// SIMATIC STEP 7 (V5.x) project KURS_PLC
// CPU: CPU 319-3 PN/DP
// station: Hardware
// station: SIMATIC 300(1)
// station: P_ADR_BUS
// program: S7 Program(2)

SYMBOL_TABLE
"SIM_M1"	DB 1	FB 1	// simulation: motor 1
"SIM_CONSTANS"	DB 2	DB 2	// simulation constants
"SIM_M"	FB 1	FB 1	// simulation: electric motor
"SIM_TANK"	FB 20	FB 20	// simulation: tank
"SIM"	FC 1	FC 1	// simulation environment
"U_TANK"	FC 20	FC 20
"h_level"	FC 21	FC 21
"U_HEAT"	FC 22	FC 22
"U_COOL"	FC 23	FC 23
"Ca"	FC 24	FC 24
"TANK"	FC 25	FC 25
"CTRL_MOTOR_SIMPLE"	FC 101	FC 101	// electric motor control
"TEST_MOTOR"	FC 1001	FC 1001	// test: CTRL_MOTOR_SIMPLE
"M1.ON"	M 1.0	BOOL
"M1.RUN"	M 1.1	BOOL
"M1.ALARM"	M 1.2	BOOL
"M1.ALARMM"	M 1.3	BOOL
"M1.RESET"	M 1.4	BOOL
"M1.CTRL"	M 1.5	BOOL
"VIN1.OPEN"	M 2.0	BOOL
"VIN1.CLOSED"	M 2.1	BOOL
"VIN2.OPEN"	M 2.2	BOOL
"VIN2.CLOSED"	M 2.3	BOOL
"k_IN1"	M 2.4	BOOL
"k_IN2"	M 2.5	BOOL
"SIM_START"	M 3.0	BOOL
"SIM_RESET"	M 3.1	BOOL
"k_HEAT"	MD 4	REAL
"k_COOL"	MD 8	REAL
"k_OUT"	MD 12	REAL
"U_COOLIN"	MD 16	REAL
"U_HEATIN"	MD 20	REAL
"U_IN2"	MD 24	REAL
"Ca_IN2"	MD 28	REAL
"U_IN1"	MD 32	REAL
"Ca_IN1"	MD 36	REAL
"Q_IN1"	MD 40	REAL
"Q_IN2"	MD 44	REAL
"SIMULATION"	OB 35	OB 35
"SRT_DINT"	SFC 32	SFC 32	// Start Time-Delay Interrupt
"QRY_DINT"	SFC 34	SFC 34	// Query Time-Delay Interrupt
"SIM_TEST"	VAT 1		// simulation test
END_SYMBOL_TABLE

FUNCTION_BLOCK "SIM_M"	// FB 1
TITLE = simulation: electric motor
//Uproszczony model silnika elektrycznego
//stany:
//STOP (0) - silnik wyłączony
//STARTING (1) - rozruch silnika
//RUN (2) - praca silnika
//STOPPING (3) - zatrzymanie silnika
VERSION : 0.1
VAR_INPUT
  On : BOOL ;	//zalaczenie silnika
  StartTime : INT ;	//czas rozruchu
  StopTime : INT ;	//czas zatrzymania
END_VAR
VAR_OUTPUT
  Run : BOOL ;
END_VAR
VAR
  State : INT ;	//numer stanu silnika
  Cnt : INT ;	//licznik czasu rozruchu/zatrzymania silnika
END_VAR
VAR_TEMP
  TempBool : BOOL ;
END_VAR
BEGIN
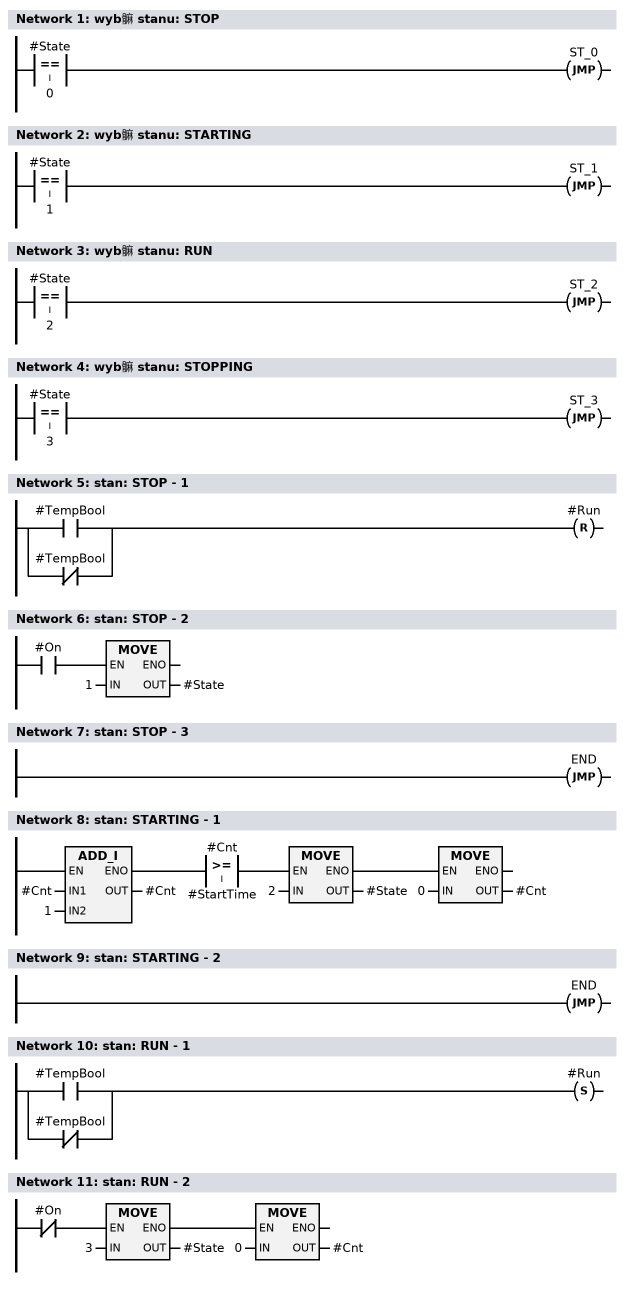
NETWORK
TITLE = wybór stanu: STOP
      L     #State;
      L     0;
      ==I;
      JC    ST_0;
NETWORK
TITLE = wybór stanu: STARTING
      L     #State;
      L     1;
      ==I;
      JC    ST_1;
NETWORK
TITLE = wybór stanu: RUN
      L     #State;
      L     2;
      ==I;
      JC    ST_2;
NETWORK
TITLE = wybór stanu: STOPPING
      L     #State;
      L     3;
      ==I;
      JC    ST_3;
NETWORK
TITLE = stan: STOP - 1
ST_0: O     #TempBool;
      ON    #TempBool;
      R     #Run;
NETWORK
TITLE = stan: STOP - 2
      A     #On;
      JNB   _001;
      L     1;
      T     #State;
_001: NOP   0;
NETWORK
TITLE = stan: STOP - 3
      JU    END;
NETWORK
TITLE = stan: STARTING - 1
ST_1: A(;
      A(;
      L     #Cnt;
      L     1;
      +I;
      T     #Cnt;
      AN    OV;
      SAVE;
      CLR;
      A     BR;
      );
      A(;
      L     #Cnt;
      L     #StartTime;
      >=I;
      );
      JNB   _002;
      L     2;
      T     #State;
      SET;
      SAVE;
      CLR;
_002: A     BR;
      );
      JNB   _003;
      L     0;
      T     #Cnt;
_003: NOP   0;
NETWORK
TITLE = stan: STARTING - 2
      JU    END;
NETWORK
TITLE = stan: RUN - 1
ST_2: O     #TempBool;
      ON    #TempBool;
      S     #Run;
NETWORK
TITLE = stan: RUN - 2
      A(;
      AN    #On;
      JNB   _004;
      L     3;
      T     #State;
      SET;
      SAVE;
      CLR;
_004: A     BR;
      );
      JNB   _005;
      L     0;
      T     #Cnt;
_005: NOP   0;
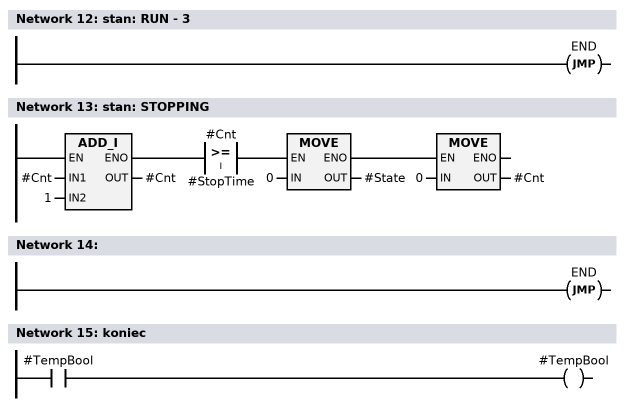
NETWORK
TITLE = stan: RUN - 3
      JU    END;
NETWORK
TITLE = stan: STOPPING
ST_3: A(;
      A(;
      L     #Cnt;
      L     1;
      +I;
      T     #Cnt;
      AN    OV;
      SAVE;
      CLR;
      A     BR;
      );
      A(;
      L     #Cnt;
      L     #StopTime;
      >=I;
      );
      JNB   _006;
      L     0;
      T     #State;
      SET;
      SAVE;
      CLR;
_006: A     BR;
      );
      JNB   _007;
      L     0;
      T     #Cnt;
_007: NOP   0;
NETWORK
TITLE =
      JU    END;
NETWORK
TITLE = koniec
END:  A     #TempBool;
      =     #TempBool;
END_FUNCTION_BLOCK

FUNCTION_BLOCK "SIM_TANK"	// FB 20
VERSION : 0.1
VAR_INPUT
  START : BOOL ;
  RESET : BOOL ;
  Q_IN1 : REAL ;
  Ca_IN1 : REAL ;
  U_IN1 : REAL ;
  Q_IN2 : REAL ;
  Ca_IN2 : REAL ;
  U_IN2 : REAL ;
  k : REAL ;
  U_HEATIN : REAL ;
  U_COOLIN : REAL ;
  NIS : INT ;
  Tc : INT ;
END_VAR
VAR
  U : REAL ;
  h : REAL ;
  Ca : REAL ;
  Ts : REAL ;
END_VAR
VAR_TEMP
  CNT : INT ;
END_VAR
BEGIN
NETWORK
TITLE = RESET
      A     #RESET;
      JCN   ERES;
      L     0.000000e+00;
      T     #U;
      L     5.000000e-01;
      T     #h;
      L     0.000000e+00;
      T     #Ca;
      L     #Tc;
      L     #NIS;
      /I;
      DTR;
      L     1.000000e+03;
      /R;
      T     #Ts;
ERES: NOP   0;
NETWORK
TITLE = SIMULATE
      AN    #RESET;
      A     #START;
      JCN   ESIM;
      L     #NIS;
      +     1;
FORJ: T     #CNT;
      CALL  "TANK" (
           Q_IN1                    := #Q_IN1,
           Ca_IN1                   := #Ca_IN1,
           U_IN1                    := #U_IN1,
           Q_IN2                    := #Q_IN2,
           Ca_IN2                   := #Ca_IN2,
           U_IN2                    := #U_IN2,
           k                        := #k,
           U_HEATIN                 := #U_HEATIN,
           U_COOLIN                 := #U_COOLIN,
           A                        := 1.000000e+00,
           h_min                    := "SIM_CONSTANS".h_min,
           k_h                      := 1.000000e+01,
           A_h                      := 1.000000e+01,
           k_c                      := 1.000000e+01,
           A_c                      := 1.000000e+01,
           Ts                       := #Ts,
           U                        := #U,
           h                        := #h,
           Ca                       := #Ca);
      L     #CNT;
      LOOP  FORJ;
ESIM: NOP   0;
END_FUNCTION_BLOCK

FUNCTION "U_TANK" : VOID	// FC 20
VERSION : 0.1
VAR_INPUT
  U_IN1 : REAL ;
  U_IN2 : REAL ;
  U_HEATIN : REAL ;
  U_COOLIN : REAL ;
  Q_IN1 : REAL ;
  Q_IN2 : REAL ;
  V : REAL ;
  h : REAL ;
  Ts : REAL ;
  k_h : REAL ;
  A_h : REAL ;
  k_c : REAL ;
  A_c : REAL ;
  h_min : REAL ;
  k : REAL ;
END_VAR
VAR_IN_OUT
  U : REAL ;
END_VAR
VAR_TEMP
  ro : REAL ;
  cw : REAL ;
  tmpCalc : REAL ;
  tmpCalc2 : REAL ;
  tmpCalc3 : REAL ;
  tmpCalc4 : REAL ;
  tmpTsV : REAL ;
  tmpRoCw : REAL ;
END_VAR
BEGIN
NETWORK
TITLE = CONSTANT
//CONSTANT
      L     1.000000e+03;
      T     #ro;
      L     4.200000e+00;
      T     #cw;
      L     #ro;
      L     #cw;
      *R;
      T     #tmpRoCw;
NETWORK
TITLE = h_min
      L     #h;
      L     #h_min;
      <R;
      JC    END;
NETWORK
TITLE =
      L     #h;
      L     "SIM_CONSTANS".h_max;
      >=R;
      JC    END;
NETWORK
TITLE = Ts/V
      L     #Ts;
      L     #V;
      /R;
      T     #tmpTsV;
NETWORK
TITLE =
      L     #Q_IN1;
      L     #U_IN1;
      *R;
      T     #tmpCalc;
      L     #Q_IN2;
      L     #U_IN2;
      *R;
      L     #tmpCalc;
      +R;
      L     #tmpTsV;
      *R;
      T     #tmpCalc;
NETWORK
TITLE =
      L     #k_h;
      L     #A_h;
      *R;
      L     #tmpTsV;
      *R;
      L     #tmpRoCw;
      /R;
      L     #U_HEATIN;
      *R;
      T     #tmpCalc2;
NETWORK
TITLE =
      L     #k_c;
      L     #A_c;
      *R;
      L     #tmpTsV;
      *R;
      L     #tmpRoCw;
      /R;
      L     #U_COOLIN;
      *R;
      T     #tmpCalc3;
NETWORK
TITLE =
// L     #k_h
//      L     #A_h
//      *R    
//      T     #tmpCalc4
//
//      L     #k_c
//      L     #A_c
//      *R    
//
//      L     #tmpCalc4
//      +R    
//      L     #tmpRoCw
//      /R    
//
//      L     #Q_IN1
//      +R    
//      L     #Q_IN2
//      +R    
//      L     #tmpTsV
//      *R    
//      L     #U
//      *R    
//      T     #tmpCalc4
//
//
//
//L     #h
//      ABS   
//      SQRT  
//      L     #k
//      *R    
//      L     #tmpTsV
//      *R    
//
      L     #Q_IN1;
      +R;
      L     #Q_IN2;
      +R;
      L     #tmpTsV;
      *R;
      L     1.000000e+00;
      TAK;
      -R;
      L     #U;
      *R;
      T     #tmpCalc4;
NETWORK
TITLE =
      L     #tmpCalc;
      L     #tmpCalc2;
      +R;
      L     #tmpCalc3;
      -R;
      L     #tmpCalc4;
      +R;
      T     #U;
NETWORK
TITLE = END
END:  NOP   0;
END_FUNCTION

FUNCTION "h_level" : VOID	// FC 21
VERSION : 0.1
VAR_INPUT
  Q_IN1 : REAL ;
  Q_IN2 : REAL ;
  k : REAL ;
  A : REAL ;
  h_max : REAL ;
  Ts : REAL ;
END_VAR
VAR_IN_OUT
  h : REAL ;
END_VAR
BEGIN
NETWORK
TITLE =
// (network holds code this reader does not know; not shown)
NETWORK
TITLE =
      L     #h;
      L     0.000000e+00;
      <R;
      JCN   Hmin;
      T     #h;
Hmin: NOP   0;
NETWORK
TITLE =
      L     #h;
      L     #h_max;
      >R;
      JCN   Hmax;
      T     #h;
Hmax: NOP   0;
END_FUNCTION

FUNCTION "U_HEAT" : VOID	// FC 22
VERSION : 0.1
VAR_INPUT
  U : REAL ;
  U_HEATIN : REAL ;
  Q_HEAT : REAL ;
  V_HEAT : REAL ;
  k_h : REAL ;
  A_h : REAL ;
  Ts : REAL ;
END_VAR
VAR_IN_OUT
  U_HEAT : REAL ;
END_VAR
VAR_TEMP
  ro : REAL ;
  cw : REAL ;
  tmpCalc : REAL ;
  tmpCalc2 : REAL ;
  tmpCalc3 : REAL ;
END_VAR
BEGIN
NETWORK
TITLE =
      L     4.200000e+03;
      T     #cw;
      L     1.000000e+03;
      T     #ro;
NETWORK
TITLE =
      L     #Ts;
      L     #V_HEAT;
      /R;
      L     #U_HEATIN;
      *R;
      L     #Q_HEAT;
      *R;
      T     #tmpCalc;
NETWORK
TITLE =
      L     #Ts;
      L     #V_HEAT;
      /R;
      L     #Q_HEAT;
      *R;
      T     #tmpCalc2;
      L     #Ts;
      L     #V_HEAT;
      /R;
      L     #k_h;
      *R;
      L     #A_h;
      *R;
      L     #ro;
      /R;
      L     #cw;
      /R;
      L     #tmpCalc2;
      +R;
      L     -1.000000e+00;
      +R;
      L     #U_HEAT;
      *R;
      T     #tmpCalc2;
NETWORK
TITLE =
      L     #Ts;
      L     #V_HEAT;
      /R;
      L     #k_h;
      *R;
      L     #A_h;
      *R;
      L     #ro;
      /R;
      L     #cw;
      /R;
      L     #U;
      *R;
      T     #tmpCalc3;
NETWORK
TITLE =
      L     #tmpCalc;
      L     #tmpCalc2;
      -R;
      L     #tmpCalc3;
      +R;
      T     #U_HEAT;
END_FUNCTION

FUNCTION "U_COOL" : VOID	// FC 23
VERSION : 0.1
VAR_INPUT
  U : REAL ;
  U_COOLIN : REAL ;
  Q_COOL : REAL ;
  V_COOL : REAL ;
  k_c : REAL ;
  A_c : REAL ;
  Ts : REAL ;
END_VAR
VAR_IN_OUT
  U_COOL : REAL ;
END_VAR
VAR_TEMP
  ro : REAL ;
  cw : REAL ;
  tmpCalc : REAL ;
  tmpCalc2 : REAL ;
  tmpCalc3 : REAL ;
END_VAR
BEGIN
NETWORK
TITLE =
      L     4.200000e+03;
      T     #cw;
      L     1.000000e+03;
      T     #ro;
NETWORK
TITLE =
      L     #Ts;
      L     #V_COOL;
      /R;
      L     #U_COOLIN;
      *R;
      L     #Q_COOL;
      *R;
      T     #tmpCalc;
NETWORK
TITLE =
      L     #Ts;
      L     #V_COOL;
      /R;
      L     #Q_COOL;
      *R;
      T     #tmpCalc2;
      L     #Ts;
      L     #V_COOL;
      /R;
      L     #k_c;
      *R;
      L     #A_c;
      *R;
      L     #ro;
      /R;
      L     #cw;
      /R;
      L     #tmpCalc2;
      TAK;
      -R;
      L     -1.000000e+00;
      +R;
      L     #U_COOL;
      *R;
      T     #tmpCalc2;
NETWORK
TITLE =
      L     #Ts;
      L     #V_COOL;
      /R;
      L     #k_c;
      *R;
      L     #A_c;
      *R;
      L     #ro;
      /R;
      L     #cw;
      /R;
      L     #U;
      *R;
      T     #tmpCalc3;
NETWORK
TITLE =
      L     #tmpCalc;
      L     #tmpCalc2;
      -R;
      L     #tmpCalc3;
      -R;
      T     #U_COOL;
END_FUNCTION

FUNCTION "Ca" : VOID	// FC 24
VERSION : 0.1
VAR_INPUT
  Q_IN1 : REAL ;
  Q_IN2 : REAL ;
  Ca_IN1 : REAL ;
  Ca_IN2 : REAL ;
  V : REAL ;
  h : REAL ;
  Ts : REAL ;
END_VAR
VAR_IN_OUT
  Ca : REAL ;
END_VAR
VAR_TEMP
  tmpCalc : REAL ;
  tmpCalc2 : REAL ;
  tmpCa : REAL ;
END_VAR
BEGIN
NETWORK
TITLE =
      L     #h;
      L     "SIM_CONSTANS".h_min;
      <R;
      JC    END;
NETWORK
TITLE =
      L     #Ca;
      T     #tmpCa;
      L     #h;
      L     "SIM_CONSTANS".h_max;
      >=R;
      JC    END;
NETWORK
TITLE =
      L     #Q_IN1;
      L     #Ca_IN1;
      *R;
      T     #tmpCalc;
      L     #Q_IN2;
      L     #Ca_IN2;
      *R;
      L     #tmpCalc;
      +R;
      L     #Ts;
      *R;
      L     #V;
      /R;
      T     #tmpCalc;
NETWORK
TITLE =
      L     #Q_IN1;
      L     #Q_IN2;
      +R;
      L     #Ts;
      *R;
      L     #V;
      /R;
      L     1.000000e+00;
      TAK;
      -R;
      L     #Ca;
      *R;
      T     #tmpCalc2;
NETWORK
TITLE =
      L     #tmpCalc;
      L     #tmpCalc2;
      +R;
      T     #Ca;
      T     #tmpCa;
NETWORK
TITLE =
END:  L     #tmpCa;
      T     #Ca;
END_FUNCTION

FUNCTION "TANK" : VOID	// FC 25
VERSION : 0.1
VAR_INPUT
  Q_IN1 : REAL ;
  Ca_IN1 : REAL ;
  U_IN1 : REAL ;
  Q_IN2 : REAL ;
  Ca_IN2 : REAL ;
  U_IN2 : REAL ;
  k : REAL ;
  U_HEATIN : REAL ;
  U_COOLIN : REAL ;
  A : REAL ;
  h_min : REAL ;
  k_h : REAL ;
  A_h : REAL ;
  k_c : REAL ;
  A_c : REAL ;
  Ts : REAL ;
END_VAR
VAR_IN_OUT
  U : REAL ;
  h : REAL ;
  Ca : REAL ;
END_VAR
VAR_TEMP
  h_p : REAL ;
  U_p : REAL ;
  V : REAL ;
  h_max : REAL ;
END_VAR
BEGIN
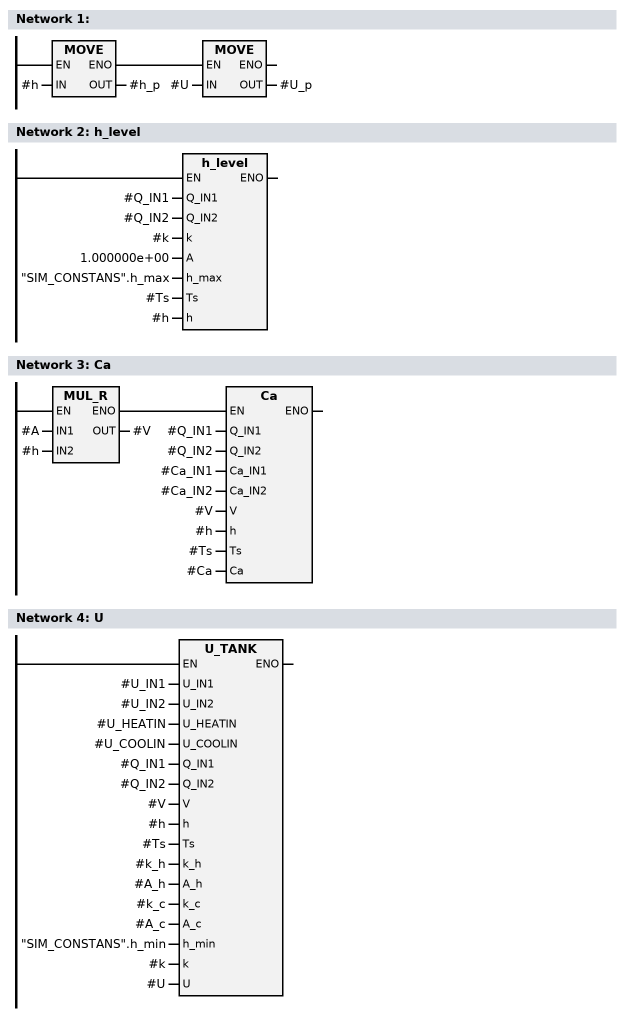
NETWORK
TITLE =
      A(;
      L     #h;
      T     #h_p;
      SET;
      SAVE;
      CLR;
      A     BR;
      );
      JNB   _001;
      L     #U;
      T     #U_p;
_001: NOP   0;
NETWORK
TITLE = h_level
      CALL  "h_level" (
           Q_IN1                    := #Q_IN1,
           Q_IN2                    := #Q_IN2,
           k                        := #k,
           A                        := 1.000000e+00,
           h_max                    := "SIM_CONSTANS".h_max,
           Ts                       := #Ts,
           h                        := #h);
      NOP   0;
NETWORK
TITLE = Ca
      A(;
      L     #A;
      L     #h;
      *R;
      T     #V;
      AN    OV;
      SAVE;
      CLR;
      A     BR;
      );
      JNB   _002;
      CALL  "Ca" (
           Q_IN1                    := #Q_IN1,
           Q_IN2                    := #Q_IN2,
           Ca_IN1                   := #Ca_IN1,
           Ca_IN2                   := #Ca_IN2,
           V                        := #V,
           h                        := #h,
           Ts                       := #Ts,
           Ca                       := #Ca);
_002: NOP   0;
NETWORK
TITLE = U
      CALL  "U_TANK" (
           U_IN1                    := #U_IN1,
           U_IN2                    := #U_IN2,
           U_HEATIN                 := #U_HEATIN,
           U_COOLIN                 := #U_COOLIN,
           Q_IN1                    := #Q_IN1,
           Q_IN2                    := #Q_IN2,
           V                        := #V,
           h                        := #h,
           Ts                       := #Ts,
           k_h                      := #k_h,
           A_h                      := #A_h,
           k_c                      := #k_c,
           A_c                      := #A_c,
           h_min                    := "SIM_CONSTANS".h_min,
           k                        := #k,
           U                        := #U);
      NOP   0;
END_FUNCTION

FUNCTION "CTRL_MOTOR_SIMPLE" : VOID	// FC 101
TITLE = control function: electric motor
VERSION : 0.1
VAR_INPUT
  On : BOOL ;	//załączenie silnika
  MotorRun : BOOL ;	//informacja o pracy silnika
  StartTimer : TIMER ;	//timer odliczający czas załączenia silnika
  StartTime : S5TIME ;	//czas trwania załączania silnika
  StopTimer : TIMER ;	//timer odmierzający czas wyłączania silnika
  StopTime : S5TIME ;	//czas trwania wyłączania silnika
  Reset : BOOL ;	//reset alarmu
END_VAR
VAR_OUTPUT
  Motor : BOOL ;	//sterowanie silnikiem
  Alarm : BOOL ;	//awaria silnika
END_VAR
VAR_IN_OUT
  AlarmM : BOOL ;
END_VAR
VAR_TEMP
  StartAlarm : BOOL ;
  StopAlarm : BOOL ;
END_VAR
BEGIN
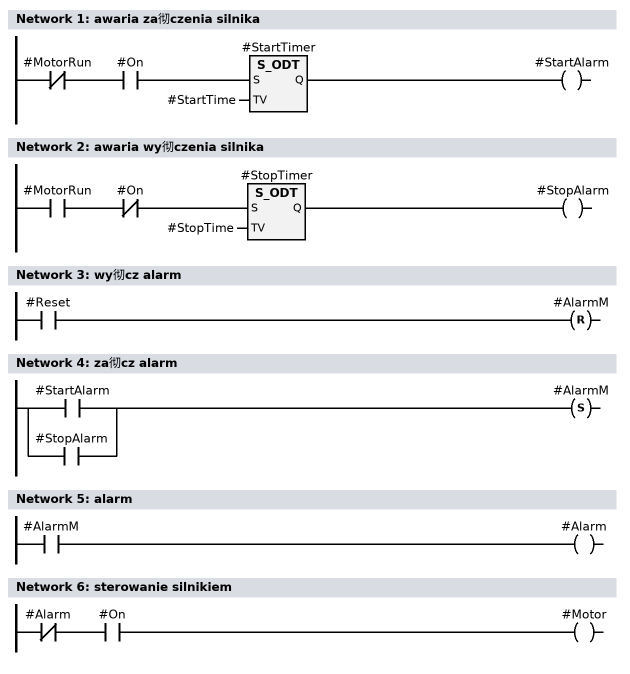
NETWORK
TITLE = awaria załączenia silnika
      AN    #MotorRun;
      A     #On;
      L     #StartTime;
      SD    #StartTimer;
      NOP   0;
      NOP   0;
      NOP   0;
      A     #StartTimer;
      =     #StartAlarm;
NETWORK
TITLE = awaria wyłączenia silnika
      A     #MotorRun;
      AN    #On;
      L     #StopTime;
      SD    #StopTimer;
      NOP   0;
      NOP   0;
      NOP   0;
      A     #StopTimer;
      =     #StopAlarm;
NETWORK
TITLE = wyłącz alarm
      A     #Reset;
      R     #AlarmM;
NETWORK
TITLE = załącz alarm
      O     #StartAlarm;
      O     #StopAlarm;
      S     #AlarmM;
NETWORK
TITLE = alarm
      A     #AlarmM;
      =     #Alarm;
NETWORK
TITLE = sterowanie silnikiem
      AN    #Alarm;
      A     #On;
      =     #Motor;
END_FUNCTION

FUNCTION "TEST_MOTOR" : VOID	// FC 1001
VERSION : 0.1
BEGIN
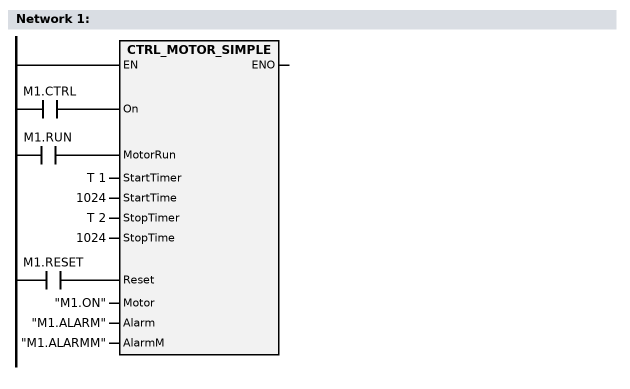
NETWORK
TITLE =
      A     "M1.CTRL";
      =     L 0.0;
      BLD   103;
      A     "M1.RUN";
      =     L 0.1;
      BLD   103;
      A     "M1.RESET";
      =     L 0.2;
      BLD   103;
      CALL  "CTRL_MOTOR_SIMPLE" (
           On                       := L 0.0,
           MotorRun                 := L 0.1,
           StartTimer               := T 1,
           StartTime                := 1024,
           StopTimer                := T 2,
           StopTime                 := 1024,
           Reset                    := L 0.2,
           Motor                    := "M1.ON",
           Alarm                    := "M1.ALARM",
           AlarmM                   := "M1.ALARMM");
      NOP   0;
END_FUNCTION

DATA_BLOCK "SIM_M1"	// DB 1
VERSION : 0.0
"SIM_M"
BEGIN
END_DATA_BLOCK

DATA_BLOCK "SIM_CONSTANS"	// DB 2
VERSION : 0.1
  STRUCT
   k_IN1_min : REAL ;	//Temporary placeholder variable
   k_IN1_max : REAL  := 2.000000e+000;	//Temporary placeholder variable
   k_IN2_min : REAL ;	//Temporary placeholder variable
   k_IN2_max : REAL  := 2.000000e+000;	//Temporary placeholder variable
   k_OUT_min : REAL ;
   k_OUT_max : REAL  := 5.000000e-001;
   U_HEATIN_min : REAL ;
   U_HEATIN_max : REAL  := 2.000000e+003;
   U_COOLIN_min : REAL ;
   U_COOLIN_max : REAL  := 2.000000e+003;
   h_min : REAL  := 5.000000e-001;
   h_max : REAL  := 1.000000e+002;
   M1StartTime : INT  := 20;	//motor no. 1 starting time
   M1StopTime : INT  := 30;	//motor no. 1 stoping time
  END_STRUCT ;	
BEGIN
   k_IN1_max := 2.000000e+00;
   k_IN2_max := 2.000000e+00;
   k_OUT_max := 5.000000e-01;
   U_HEATIN_max := 2.000000e+03;
   U_COOLIN_max := 2.000000e+03;
   h_min := 5.000000e-01;
   h_max := 1.000000e+02;
   M1StartTime := 70;
   M1StopTime := 30;
END_DATA_BLOCK

DATA_BLOCK DB 20
VERSION : 0.0
"SIM_TANK"
BEGIN
END_DATA_BLOCK

ORGANIZATION_BLOCK OB 1
TITLE = "Main Program Sweep (Cycle)"
VERSION : 0.1
VAR_TEMP
  OB1_EV_CLASS : BYTE ;	//Bits 0-3 = 1 (Coming event), Bits 4-7 = 1 (Event class 1)
  OB1_SCAN_1 : BYTE ;	//1 (Cold restart scan 1 of OB 1), 3 (Scan 2-n of OB 1)
  OB1_PRIORITY : BYTE ;	//Priority of OB Execution
  OB1_OB_NUMBR : BYTE ;	//1 (Organization block 1, OB1)
  OB1_RESERVED_1 : BYTE ;	//Reserved for system
  OB1_RESERVED_2 : BYTE ;	//Reserved for system
  OB1_PREV_CYCLE : INT ;	//Cycle time of previous OB1 scan (milliseconds)
  OB1_MIN_CYCLE : INT ;	//Minimum cycle time of OB1 (milliseconds)
  OB1_MAX_CYCLE : INT ;	//Maximum cycle time of OB1 (milliseconds)
  OB1_DATE_TIME : DATE_AND_TIME ;	//Date and time OB1 started
END_VAR
BEGIN
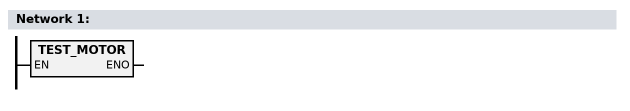
NETWORK
TITLE =
      CALL  "TEST_MOTOR";
      NOP   0;
END_ORGANIZATION_BLOCK

ORGANIZATION_BLOCK "SIMULATION"	// OB 35
TITLE = "Cyclic Interrupt"
VERSION : 0.1
VAR_TEMP
  OB35_EV_CLASS : BYTE ;	//Bits 0-3 = 1 (Coming event), Bits 4-7 = 1 (Event class 1)
  OB35_STRT_INF : BYTE ;	//16#36 (OB 35 has started)
  OB35_PRIORITY : BYTE ;	//Priority of OB Execution
  OB35_OB_NUMBR : BYTE ;	//35 (Organization block 35, OB35)
  OB35_RESERVED_1 : BYTE ;	//Reserved for system
  OB35_RESERVED_2 : BYTE ;	//Reserved for system
  OB35_PHASE_OFFSET : WORD ;	//Phase offset (msec)
  OB35_RESERVED_3 : INT ;	//Reserved for system
  OB35_EXC_FREQ : INT ;	//Frequency of execution (msec)
  OB35_DATE_TIME : DATE_AND_TIME ;	//Date and time OB35 started
END_VAR
BEGIN
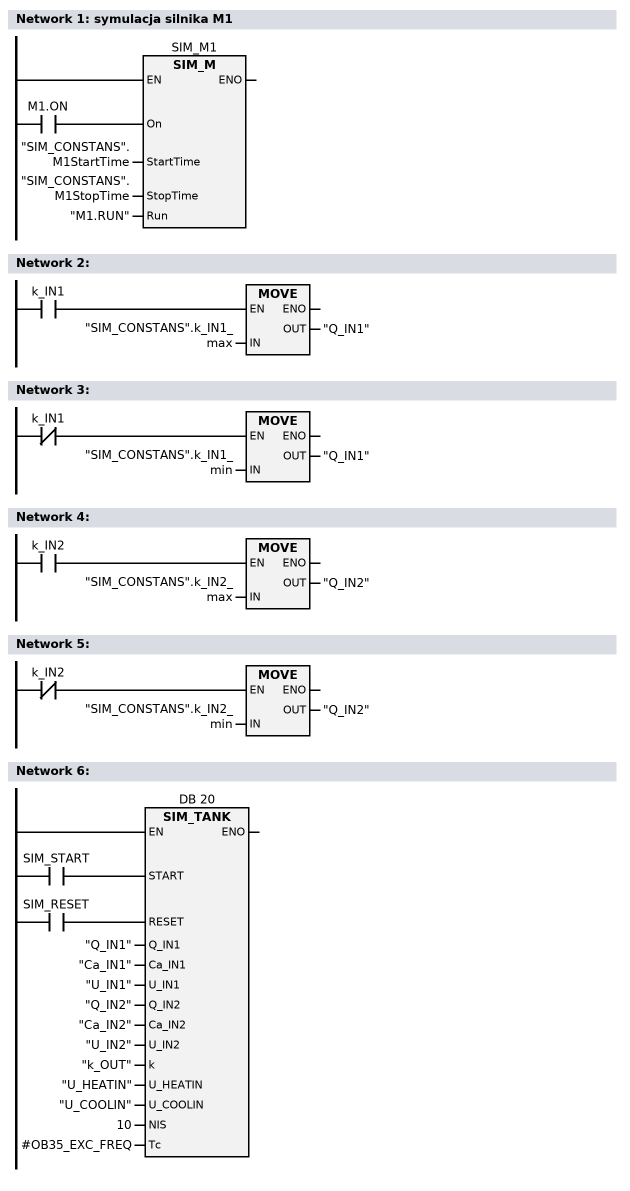
NETWORK
TITLE = symulacja silnika M1
      A     "M1.ON";
      =     L 20.0;
      BLD   103;
      CALL  "SIM_M" , "SIM_M1" (
           On                       := L 20.0,
           StartTime                := "SIM_CONSTANS".M1StartTime,
           StopTime                 := "SIM_CONSTANS".M1StopTime,
           Run                      := "M1.RUN");
      NOP   0;
NETWORK
TITLE =
      A     "k_IN1";
      JNB   _001;
      L     "SIM_CONSTANS".k_IN1_max;
      T     "Q_IN1";
_001: NOP   0;
NETWORK
TITLE =
      AN    "k_IN1";
      JNB   _002;
      L     "SIM_CONSTANS".k_IN1_min;
      T     "Q_IN1";
_002: NOP   0;
NETWORK
TITLE =
      A     "k_IN2";
      JNB   _003;
      L     "SIM_CONSTANS".k_IN2_max;
      T     "Q_IN2";
_003: NOP   0;
NETWORK
TITLE =
      AN    "k_IN2";
      JNB   _004;
      L     "SIM_CONSTANS".k_IN2_min;
      T     "Q_IN2";
_004: NOP   0;
NETWORK
TITLE =
      A     "SIM_START";
      =     L 20.0;
      BLD   103;
      A     "SIM_RESET";
      =     L 20.1;
      BLD   103;
      CALL  "SIM_TANK" , DB 20 (
           START                    := L 20.0,
           RESET                    := L 20.1,
           Q_IN1                    := "Q_IN1",
           Ca_IN1                   := "Ca_IN1",
           U_IN1                    := "U_IN1",
           Q_IN2                    := "Q_IN2",
           Ca_IN2                   := "Ca_IN2",
           U_IN2                    := "U_IN2",
           k                        := "k_OUT",
           U_HEATIN                 := "U_HEATIN",
           U_COOLIN                 := "U_COOLIN",
           NIS                      := 10,
           Tc                       := #OB35_EXC_FREQ);
      NOP   0;
NETWORK
TITLE =
END_ORGANIZATION_BLOCK
